# EPICS substitutions: example/exampleApp/Db/example.substitutions
file OXCS700.template
{
pattern { P      , Q , PORT    }
        { OXCS700, "", OXCS700p }
}

file OXPH700.template
{
pattern { P      , Q , PORT    }
        { OXPH700, "", OXPH700p }
}
